PROGRAM PRG_Tests
VAR
  testRunner : T_TestRunner;
  
  //Modes
  modeTestSuite : T_TestSuite;
  ProductionToMaintenaceInAbort : T_ProductionToMaintenaceInAbort(modeTestSuite);
  CantChangeModInExecute : T_CantChangeModInExecute(modeTestSuite);
  JogThroughStates : T_JogThroughStates(modeTestSuite);
  CantChangeStateFromIdleToSuspend : T_CantChangeStateFromIdleToSuspend(modeTestSuite);
  
  // set mode
  AddPackModeSetsCorrectly : T_AddPackModeSetsCorrectly(modeTestSuite);  
  InitModeManagerWithState : T_InitModeManagerWithState(modeTestSuite);
  ModeChangeFromProductionToMaintenance : T_ModeChangeFromProductionToMaintenance(modeTestSuite);
  ModeInitialisedFromInvalidToProduction : T_ModeInitialisedFromInvalidToProduction(modeTestSuite);
  
  
END_VAR

IF testRunner.ReloadTests THEN
    testRunner.AddTestSuite(modeTestSuite);
    testRunner.ReloadTests := FALSE;
END_IF

testRunner();

END_PROGRAM

(* stored: Version 1.1.0.1, ProductVersion 3.1.4024.12
   POU PRG_Tests: Id {5e432f02-8359-43cd-91aa-bd5cdb5f4243}, SpecialFunc None *)
